// TIA Portal V21 export
TYPE "Std_Pid"
   STRUCT
      In : Struct
         ChiudiPid : Bool;
         ApriPid : Bool;
         "%ApriPid" : Real;
         EsclusioneAllarmi : Bool;
         EnLimitaMinUscita : Bool;
         EnLimitaMaxUscita : Bool;
         LimitaMinUscita : Bool;
         LimitaMaxUscita : Bool;
         K_Motore1 : Int;
         K_Motore2 : Int;
         K_Valvola1 : Int;
         K_Valvola2 : Int;
         K_Analogica_Uscita : Int;   // La mia uscita attuale viene passata alla gestione analogica
      END_STRUCT;
      Prm : Struct
         MinOut : Real;   // Minima uscita del PID durante funzionamento automatico
         MaxOut : Real := 100.0;   // Massima uscita del PID durante funzionamento automatico
         LimitMinOut : Real;   // Se abilitata e se richiesta limita la minima uscita del PID
         LimitMaxOut : Real;   // Se abilitata e se richiesta limita la massima uscita del PID
         EnResettaComponenti : Bool;   // Abilitazione al reset delle componenti
         ResettaComponentiConCmdMan : Bool;
         PermettiCadutaCicloAutomatico : Bool;
         ComandaUtenzaInUscita : Bool;
         K_TipoAccoppiamentoUscitePid : Int;
         DeadbandAccoppiamentoUscite : Real;
         RampaSetpoint : Struct
            Abilitazione : Bool;
            RampUpRate : Real;
            RampDownRate : Real;
         END_STRUCT;
         UnitàMisura : "Std_UnitàDiMisura";
         FF : Struct
            interpolazione : Array[0..20] of Struct
               Setpoint : Real;
               Valore : Real;
            END_STRUCT;
            RicercaValore : Struct
               Abilitazione : Bool := FALSE;
               UscitaDiComando : Real := -2.6;
            END_STRUCT;
         END_STRUCT;
         BIAS : Struct
            DeadBand : Real := 0.3;
            MaxLimit_Out : Real := 10.0;
            MinLimit_Out : Real := -10.0;
            KCorr : Real := 0.0009943267;
            K : Real := 0.0012;
         END_STRUCT;
         EquilibriumSeeking : Struct   // Ricerca periodica del punto di contatto
            FrequenzaAvvioTest : "Std_stTimer";   // Ogni quanto viene ripetuto il test
            TimeoutRicerca { S7_SetPoint := 'True'} : "Std_stTimer";   // Tempo in cui devo raggiungere la variazione sul setpoint, altrimenti si blocca
            DurataGradinoVariazione : "Std_stTimer";   // Per quanto tempo aspetto la reazione del sistema
            DurataVariazioneAnalogica { S7_SetPoint := 'True'} : "Std_stTimer";
            VariazioneMinimaAnalogica { S7_SetPoint := 'True'} : Real := 1.0;   // Variazione minima che devo vedere sul setpoint
            DirezioneRicercaPos : Bool := False;   // 1 = La ricerca avviene in direzione positiva 0 = Negativa
            VariazioneSulComando : Real := 0.5;   // Di quanto cambio il comando ad ogni gradino
         END_STRUCT;
      END_STRUCT;
      Hmi : Struct
         Man : Bool;
         Auto : Bool;
         Stop : Bool;
         ReinizzializzaComponenti : Bool;
         ValoreIntegraleAttuale : Real;
         ValoreDerivataAttuale : Real;
         Sp_Ki : Real;
         Sp_Kd : Real;
         Sp_Kp : Real;
         AttualeRifAnalog : Real;
         InversionePid : Bool;
         SetpointPID : Real;
         SetpointFF : Real;   // Setpoint da inseguire con il FF
         SetpointFF_DaPid : Bool := True;   // Il setpoint del FF viene copiato dal PID
         InterpolazioniFF : Struct
            IndiceHmiPrec : Int;
            IndiceHmi : Int;
            Setpoint : Real;
            Valore : Real;
         END_STRUCT;
         StatoUscitaPID : Real;
         Erorre : Real;
         AperturaManReq : Real;
         AvviaAutoTuning : Bool;
         AutotuningRichiesto : Bool;
         AutotuningInCorso : Bool;
         AutotuningProgress : Real;
         Diagnostica : Struct
            "0-PIDForzatoChiusoDaPlc" : Bool;
            "1-PIDForzatoApertoDaPlc" : Bool;
            "2-PidChiusoCausaCicloAutomatico" : Bool;
            "3-AllarmiPidEsclusi" : Bool;
            "4-ResetIntegraleInCorso" : Bool;
            "5-SuperamentoMassimoSp" : Bool;
            "6-SuperamentoMinimoSp" : Bool;
            "7-TroppoTempoFuoriSetpoint" : Bool;
            "8-LimiteMinimaUscitaPIDRichiestaPlc" : Bool;
            "9-LimiteMassimaUscitaPIDRichiestaPlc" : Bool;
            "10-UtenzaInUscitaInStop" : Bool;
            "11-EquilibriumSeekingInCorso" : Bool;
            "12-AutotuningInCorso" : Bool;
         END_STRUCT;
         VisualizzazioniHMI : Struct
            LimiteMinimaUscita : Bool;
            LimiteMassimaUscita : Bool;
            VisualizzaRampaSetpoint : Bool;
         END_STRUCT;
         AbilitazionePID : Bool;
         AbilitazioneFF : Bool;
         AbilitazioneBIAS : Bool;
         AbilitazioneEquilibriumSeeking : Bool;
      END_STRUCT;
      Dati : Struct
         SetpointPrecedente : Real;
         ModePrecedente : Int;   // Stato del parametro mode nello stato precedente
         AttendiTermineAutotuning : Bool;
         ReinizializzaComponenti : Bool;
         EquilibriumSeeking : Struct
            InCorso : Bool;
            Setpoint : Real;
         END_STRUCT;
         StabilizzazioneSetpoint : Struct
            Setpoint_Precedente : Real := 40.0;
            SetpointStabile_Preset : Int := 100;
            SetpointStabile_Attuale : Int := -30605;
            Setpoint_Discesa : Bool := TRUE;
            Setpoint_Salita : Bool := FALSE;
            SetpointStabile_Raggiunto : Bool := FALSE;
         END_STRUCT;
         StabilizzazioneAnalogica : Struct
            Attuale_Precedente : Real := 0.0;
            AttualeStabile_Preset : Int := 250;
            AttualeStabile_Attuale : Int := 27020;
            Attuale_Discesa : Bool := TRUE;
            Attuale_Salita : Bool := FALSE;
            AttualeStabile_Raggiunto : Bool := TRUE;
         END_STRUCT;
         Errore : Real := 40.0;
         UltimoErroreMedioNelTempo : Real := 40.0;
         SommaErroreNelTempo : Real := 3240.0;
         NumeroMedieCalcolte : Real := 81.0;
      END_STRUCT;
      Allarmi : Struct
         "Timer" : "Std_stTimer";
         PresetSoglie { S7_SetPoint := 'True'} : "Std_Pid_Allarmi";
         "A" : Array[0.."K_NumAllarmiPerPid"] of "Std_PrmAllarmeStd";
         WordHMI { S7_SetPoint := 'True'} : Word;
      END_STRUCT;
      Out : Struct
         Uscita_DaPid : Real := 0.0;
         Uscita_DaFF : Real := -1.990769;
         Uscita_DaBIAS : Real := 0.0;
         TotaleUscitaAttuale : Real := -1.990769;
         VelRichiestaMotore : Int;
         Paw : Int;
      END_STRUCT;
      Rif_Inc : Struct
         K_Analogica : Int;
         K_Motore1 : Int;
         K_Motore2 : Int;
         K_Valvola1 : Int;
         K_Valvola2 : Int;
         K_Zona : Int;
         K_Analogica_Uscita : Int;
      END_STRUCT;
   END_STRUCT;
   // Prm.UnitàMisura.Out.UmCode := 3;
   // Prm.EquilibriumSeeking.FrequenzaAvvioTest.Preset := 300.0;
   // Prm.EquilibriumSeeking.TimeoutRicerca.Preset := 120.0;
   // Prm.EquilibriumSeeking.DurataGradinoVariazione.Preset := 1.0;
   // Prm.EquilibriumSeeking.DurataVariazioneAnalogica.Preset := 1.0;
   // // Allarmi."A"[1] : MinSetPoint
   // // Allarmi."A"[2] : MaxSetPoint
   // // Allarmi."A"[3] : TroppoTempoAllarme
END_TYPE
